Staubli VAL3: onF8Event.pgx

program onF8Event(bool& x_bSave[])
  local num i
begin
  // look if the bButton is enable
  if bButton[7]
    //
    call saveIt(x_bSave)
  endIf
end
